(* IEC 61131-3 sources: TrakMap/InstallerSetup/Installer AS Technology Solution/Logical/Source/Diagnostic/TrakDiag, 7 files *)

(* ---- Types.typ ---- *)
TYPE
	VisType : 	STRUCT
		OpenSegDialog : BOOL;
		OpenShuttleDialog : BOOL;
	END_STRUCT;
	CheckStateEnum :
		(
		WAIT_FOR_CHECK,
		READ_DATA,
		READ_DATA_SEG_STATE,
		CHECK_SEG_STATE,
		READ_DATA_SEG_ERROR_STAT,
		CHECK_ERROR_STAT,
		READ_DATA_SEG_ERROR,
		CHECK_ERROR_CODE,
		WRITE_WARNING_CODE,
		READ_DATA_SEG_LAG,
		CHECK_SEG_LAG,
		READ_DATA_SEG_VEL,
		CHECK_SEG_VEL,
		READ_DATA_SEG_TEMP,
		CHECK_DATA_SEG_TEMP,
		WRITE_SPEED_FILTER,
		WRITE_SPEED_FILTER_WAIT,
		WRITE_ZERO_PITCH,
		READ_EXEC_ERROR,
		READ_SEG_STATUS,
		WRITE_SEG_RESET,
		WAIT_FOR_DONE
		);
	SegErrorCheckType : 	STRUCT
		CheckState : CheckStateEnum;
		CmdCheckErrorCode : BOOL;
		DataReadExecutionError : BOOL;
		ErrorNumber : UINT;
		SegStatusBits : UDINT;
		ErrorStatusBit : BOOL;
		ErrorStatus : UDINT;
	END_STRUCT;
	DiagFbsType : 	STRUCT
		Asm : DiagAsmFbsTyp;
		Seg : DiagSegFbsTyp;
	END_STRUCT;
	DiagAsmFbsTyp : 	STRUCT
		ReadInfo : MC_BR_AsmReadInfo_AcpTrak;
		ReadStatus : MC_BR_AsmReadStatus_AcpTrak;
	END_STRUCT;
	DiagSegFbsTyp : 	STRUCT
		ReadInfo : ARRAY[0..NUM_SEG]OF MC_BR_SegReadInfo_AcpTrak;
		ReadStatus : ARRAY[0..NUM_SEG]OF MC_BR_SegReadStatus_AcpTrak;
		ProcessParID : ARRAY[0..NUM_SEG]OF MC_BR_SegProcessParID_AcpTrak;
	END_STRUCT;
END_TYPE

(* ---- CheckErrorCode.st ---- *)
ACTION actCheckErrorCode:

	FOR SegIndex := 0 TO NUM_SEG DO

		CASE SegErrorCheck[SegIndex].CheckState OF

			WAIT_FOR_CHECK:
				//Wait for the command to check the error code ParID on the segment
				DiagFbs.Seg.ProcessParID[SegIndex].Execute := FALSE;

				IF SegErrorCheck[SegIndex].CmdCheckErrorCode THEN
					ErrorCodeIDInfo[SegIndex].DataType := mcACPTRAK_SEG_PARTYPE_UINT;
					ErrorCodeIDInfo[SegIndex].ParID := mcACPPAR_ERROR_NUMBER;
					ErrorCodeIDInfo[SegIndex].VariableAddress := ADR(SegErrorCheck[SegIndex].ErrorNumber);

					DiagFbs.Seg.ProcessParID[SegIndex].Execute := TRUE;
					DiagFbs.Seg.ProcessParID[SegIndex].Segment := ADR(TrakDiag.Seg.SegList[SegIndex].McType);
					DiagFbs.Seg.ProcessParID[SegIndex].ChannelIndex := 0;
					DiagFbs.Seg.ProcessParID[SegIndex].NumberOfParIDs := 1;
					DiagFbs.Seg.ProcessParID[SegIndex].Mode := mcACPTRAK_SEG_PARID_GET_NO_NCT;
					DiagFbs.Seg.ProcessParID[SegIndex].DataAddress := ADR(ErrorCodeIDInfo[SegIndex]);
					SegErrorCheck[SegIndex].CheckState := READ_DATA_SEG_ERROR;
					SegErrorCheck[SegIndex].CmdCheckErrorCode := FALSE; //Reset check command

				END_IF

			READ_DATA_SEG_ERROR:
				//Check for completion of reading the PARID for

				IF DiagFbs.Seg.ProcessParID[SegIndex].Done THEN
					//If the parID was successfully read, go to check error code state
					SegErrorCheck[SegIndex].CheckState := CHECK_ERROR_CODE;
					DiagFbs.Seg.ProcessParID[SegIndex].Execute := FALSE;
					SegErrorCheck[SegIndex].DataReadExecutionError := FALSE;

				ELSIF DiagFbs.Seg.ProcessParID[SegIndex].Error THEN
					//If there was an error in reading, go to error start
					SegErrorCheck[SegIndex].CheckState := READ_EXEC_ERROR;
				END_IF
			CHECK_ERROR_CODE:

				IF (SegErrorCheck[SegIndex].ErrorNumber = 0) OR (SegErrorCheck[SegIndex].ErrorNumber = 36005) THEN
					//Segment has no new error recorded. Shows either 0 or the commanded warning (36005) used to overwrite old errors
					TrakDiag.Seg.SegList[SegIndex].Status.ErrorCode := 0;
					SegErrorCheck[SegIndex].CheckState := WAIT_FOR_CHECK;
					TrakDiag.Seg.SegList[SegIndex].Status.Error := FALSE;

				ELSE
					//Otherwise, there is a new error on this segment
					TrakDiag.Seg.SegList[SegIndex].Status.ErrorCode := SegErrorCheck[SegIndex].ErrorNumber;

					TrakDiag.Seg.SegList[SegIndex].Status.Error := TRUE;
					//Send to overwrite state to store a known error number (36005) in the error code parID
					SegErrorCheck[SegIndex].CheckState := WRITE_WARNING_CODE;

				END_IF
			WRITE_WARNING_CODE:
				//Write commanded warning code (36005) to error parid
				DiagFbs.Seg.ProcessParID[SegIndex].DataAddress := ADR(SegWarningCmdIDInfo);
				DiagFbs.Seg.ProcessParID[SegIndex].ChannelIndex := 0;
				DiagFbs.Seg.ProcessParID[SegIndex].Mode := mcACPTRAK_SEG_PARID_SET;
				DiagFbs.Seg.ProcessParID[SegIndex].NumberOfParIDs := 0;
				DiagFbs.Seg.ProcessParID[SegIndex].Execute := TRUE;

				IF DiagFbs.Seg.ProcessParID[SegIndex].Done THEN
					//return to wait state
					DiagFbs.Seg.ProcessParID[SegIndex].Execute := FALSE;
					SegErrorCheck[SegIndex].CheckState := WAIT_FOR_CHECK;

				ELSIF DiagFbs.Seg.ProcessParID[SegIndex].Error THEN
					SegErrorCheck[SegIndex].CheckState := READ_EXEC_ERROR;
				END_IF
			READ_EXEC_ERROR:
				DiagFbs.Seg.ProcessParID[SegIndex].Execute := FALSE;
				SegErrorCheck[SegIndex].DataReadExecutionError := TRUE;

				IF DiagFbs.Seg.ProcessParID[SegIndex].Error = FALSE THEN
					SegErrorCheck[SegIndex].CheckState := WAIT_FOR_CHECK;
				END_IF
		END_CASE
	DiagFbs.Seg.ProcessParID[SegIndex]();
	END_FOR
END_ACTION

(* ---- Cyclic.st ---- *)
PROGRAM _CYCLIC

	MC_BR_SegCommandError_AcpTrak_0(Segment := ADR(TrakDiag.Seg.SegList[0].McType));

	IF MC_BR_SegCommandError_AcpTrak_0.Done THEN
		MC_BR_SegCommandError_AcpTrak_0.Execute := FALSE;
	END_IF

	(***********************************ASSEMBLY INFORMATION******************************	)
	(*Read Assebly Status*)

	DiagFbs.Asm.ReadStatus.Enable	:= TRUE;
	DiagFbs.Asm.ReadStatus();

	IF DiagFbs.Asm.ReadStatus.Valid THEN
		TrakDiag.Asm.AssemblyDisabled 	:= DiagFbs.Asm.ReadStatus.AssemblyDisabled;
		TrakDiag.Asm.AssemblyErrorStop := DiagFbs.Asm.ReadStatus.AssemblyErrorStop;
		TrakDiag.Asm.AssemblyReady		:= DiagFbs.Asm.ReadStatus.AssemblyReady;
		TrakDiag.Asm.AssemblyHoming	:= DiagFbs.Asm.ReadStatus.AssemblyHoming;
		TrakDiag.Asm.AssemblyStopping	:= DiagFbs.Asm.ReadStatus.AssemblyStopping;
	END_IF

	(*Read Assembly Info *)

	DiagFbs.Asm.ReadInfo.Enable		:= TRUE;
	DiagFbs.Asm.ReadInfo();

	IF DiagFbs.Asm.ReadInfo.Valid THEN
		TrakDiag.Asm.CommunicationReady 	:= DiagFbs.Asm.ReadInfo.AssemblyInfo.CommunicationReady;
		TrakDiag.Asm.PowerOn				:= DiagFbs.Asm.ReadInfo.AssemblyInfo.PowerOn;
		TrakDiag.Asm.ReadyForPowerOn		:= DiagFbs.Asm.ReadInfo.AssemblyInfo.ReadyForPowerOn;
		TrakDiag.Asm.ShuttlesCount 			:= DiagFbs.Asm.ReadInfo.AssemblyInfo.ShuttlesCount;
		TrakDiag.Asm.ShuttleInErrorStopCount := DiagFbs.Asm.ReadInfo.AssemblyInfo.ShuttlesInErrorStopCount;
		TrakDiag.Asm.StartupCount			:= DiagFbs.Asm.ReadInfo.AssemblyInfo.StartupCount;
	END_IF

	(****************************** SEGMENT ERROR INFORMATION *****************************************)

	FOR SegIndex := 0 TO NUM_SEG DO

		IF TrakDiag.Seg.SegList[SegIndex].McType.controlif <> 0 THEN //If the array contains a segment reference

			DiagFbs.Seg.ReadInfo[SegIndex].Segment 	:= ADR(TrakDiag.Seg.SegList[SegIndex].McType);
			DiagFbs.Seg.ReadInfo[SegIndex].Enable	:= TRUE;
			DiagFbs.Seg.ReadInfo[SegIndex]();

			IF DiagFbs.Seg.ReadInfo[SegIndex].Valid THEN
				//Capture Segment Info
				TrakDiag.Seg.SegList[SegIndex].Status.CommunicationReady 	:= DiagFbs.Seg.ReadInfo[SegIndex].SegmentInfo.CommunicationReady;
				TrakDiag.Seg.SegList[SegIndex].Status.ReadyForPowerOn		:= DiagFbs.Seg.ReadInfo[SegIndex].SegmentInfo.ReadyForPowerOn;
				TrakDiag.Seg.SegList[SegIndex].Status.PowerOn				:= DiagFbs.Seg.ReadInfo[SegIndex].SegmentInfo.PowerOn;
				TrakDiag.Seg.SegList[SegIndex].Status.StartupCount			:= DiagFbs.Seg.ReadInfo[SegIndex].SegmentInfo.StartupCount;
				TrakDiag.Seg.SegList[SegIndex].Status.CommunicationState	:= DiagFbs.Seg.ReadInfo[SegIndex].SegmentInfo.CommunicationState;

			END_IF

			DiagFbs.Seg.ReadStatus[SegIndex].Segment := ADR(TrakDiag.Seg.SegList[SegIndex].McType);
			DiagFbs.Seg.ReadStatus[SegIndex].Enable	:= TRUE;
			DiagFbs.Seg.ReadStatus[SegIndex]();

			IF DiagFbs.Seg.ReadStatus[SegIndex].Valid THEN

				//Check for change of state to ErrorStop to command reading error data, IF communication is ready
				IF ((TrakDiag.Seg.SegList[SegIndex].Status.SegmentErrorStop = FALSE AND DiagFbs.Seg.ReadStatus[SegIndex].SegmentErrorStop = TRUE))
					AND (TrakDiag.Seg.SegList[SegIndex].Status.CommunicationReady = TRUE) THEN

					SegErrorCheck[SegIndex].CmdCheckErrorCode := TRUE;

					//Check for change of state from ErrorStop to reset error number in diag structure
				ELSIF ((TrakDiag.Seg.SegList[SegIndex].Status.SegmentErrorStop = TRUE) AND (DiagFbs.Seg.ReadStatus[SegIndex].SegmentErrorStop = FALSE))
					AND (TrakDiag.Seg.SegList[SegIndex].Status.CommunicationReady = TRUE) THEN

					TrakDiag.Seg.SegList[SegIndex].Status.ErrorCode := 0;

				END_IF
				//Capture Segment Status

				TrakDiag.Seg.SegList[SegIndex].Status.SegmentDisabled	:= DiagFbs.Seg.ReadStatus[SegIndex].SegmentDisabled;
				TrakDiag.Seg.SegList[SegIndex].Status.SegmentErrorStop	:= DiagFbs.Seg.ReadStatus[SegIndex].SegmentErrorStop;
				TrakDiag.Seg.SegList[SegIndex].Status.SegmentReady		:= DiagFbs.Seg.ReadStatus[SegIndex].SegmentReady;
				TrakDiag.Seg.SegList[SegIndex].Status.SegmentStopping	:= DiagFbs.Seg.ReadStatus[SegIndex].SegmentStopping;
			END_IF
		END_IF
	END_FOR

	CpuSim := DiagCpuIsSimulated() OR DiagCpuIsARsim();

	IF CpuSim = FALSE THEN
		actCheckErrorCode;
	END_IF

	(***********************************TRAKMAP******************************)

	//Fetch ShuttleUserData Example
	IF EDGEPOS(paperCore.ClickData.Shuttle.Valid) THEN
		MC_BR_ShCopyUserData_AcpTrak_0.Axis         := ADR(paperCore.ClickData.Shuttle.Data.Axis);
		MC_BR_ShCopyUserData_AcpTrak_0.Execute      := TRUE;
		MC_BR_ShCopyUserData_AcpTrak_0.DataAddress  := ADR(ShuttleUserData);
		MC_BR_ShCopyUserData_AcpTrak_0.DataSize     := SIZEOF(ShuttleUserData);
		MC_BR_ShCopyUserData_AcpTrak_0.Mode         := mcACPTRAK_USERDATA_GET;
	END_IF

	paperCore();

	MC_BR_ShCopyUserData_AcpTrak_0();
	MC_BR_ShCopyUserData_AcpTrak_0.Execute := FALSE;

END_PROGRAM

(* ---- Exit.st ---- *)
PROGRAM _EXIT
			(* Insert code here *)

END_PROGRAM

(* ---- Init.st ---- *)
PROGRAM _INIT

	SegDefinition;

	paperCore.SegmentCount := TrakDiag.Seg.SegCount;
	paperCore.Segments := ADR(TrakDiag.Seg.SegList);
	paperCore.Options := ADR(paperOptions);
	paperCore.Enable := TRUE;
	paperCore.Assembly := ADR(DiagInterface.SampleTrak);
	paperCore.ShuttleMon := ADR(DiagInterface.ShuttleMon);
	paperCore.TrakStatus := ADR(TrakDiag);

	paperOptions.Color.Offset := SIZEOF(UDINT);
	paperOptions.Segment.Enabled := TRUE;
	paperOptions.Shuttle.Enabled := TRUE;
	paperOptions.Color.Enabled := TRUE;
END_PROGRAM

(* ---- SegDefinition.st ---- *)
//This file was automatically generated using the TrakMapImporter program. Verify that the segment names and assembly name match your project values correctly
ACTION SegDefinition:
	TrakDiag.Seg.SegList[0].Name  := 'gSeg_A_1';		TrakDiag.Seg.SegList[0].McType := gSeg_A_1;
	TrakDiag.Seg.SegList[1].Name  := 'gSeg_A_2';		TrakDiag.Seg.SegList[1].McType := gSeg_A_2;
	TrakDiag.Seg.SegList[2].Name  := 'gSeg_A_3';		TrakDiag.Seg.SegList[2].McType := gSeg_A_3;
	TrakDiag.Seg.SegList[3].Name  := 'gSeg_A_4';		TrakDiag.Seg.SegList[3].McType := gSeg_A_4;
	TrakDiag.Seg.SegList[4].Name  := 'gSeg_A_5';		TrakDiag.Seg.SegList[4].McType := gSeg_A_5;
	TrakDiag.Seg.SegList[5].Name  := 'gSeg_A_6';		TrakDiag.Seg.SegList[5].McType := gSeg_A_6;
	TrakDiag.Seg.SegList[6].Name  := 'gSeg_A_7';		TrakDiag.Seg.SegList[6].McType := gSeg_A_7;
	TrakDiag.Seg.SegList[7].Name  := 'gSeg_A_8';		TrakDiag.Seg.SegList[7].McType := gSeg_A_8;
	TrakDiag.Seg.SegList[8].Name  := 'gSeg_A_9';		TrakDiag.Seg.SegList[8].McType := gSeg_A_9;
	TrakDiag.Seg.SegList[9].Name  := 'gSeg_A_10';		TrakDiag.Seg.SegList[9].McType := gSeg_A_10;
	TrakDiag.Seg.SegList[10].Name  := 'gSeg_A_11';		TrakDiag.Seg.SegList[10].McType := gSeg_A_11;
	TrakDiag.Seg.SegList[11].Name  := 'gSeg_A_12';		TrakDiag.Seg.SegList[11].McType := gSeg_A_12;

	TrakDiag.Seg.SegList[12].Name  := 'gSeg_B_1';		TrakDiag.Seg.SegList[12].McType := gSeg_B_1;
	TrakDiag.Seg.SegList[13].Name  := 'gSeg_B_2';		TrakDiag.Seg.SegList[13].McType := gSeg_B_2;
	TrakDiag.Seg.SegList[14].Name  := 'gSeg_B_3';		TrakDiag.Seg.SegList[14].McType := gSeg_B_3;
	TrakDiag.Seg.SegList[15].Name  := 'gSeg_B_4';		TrakDiag.Seg.SegList[15].McType := gSeg_B_4;
	TrakDiag.Seg.SegList[16].Name  := 'gSeg_B_5';		TrakDiag.Seg.SegList[16].McType := gSeg_B_5;
	TrakDiag.Seg.SegList[17].Name  := 'gSeg_B_6';		TrakDiag.Seg.SegList[17].McType := gSeg_B_6;
	TrakDiag.Seg.SegList[18].Name  := 'gSeg_B_7';		TrakDiag.Seg.SegList[18].McType := gSeg_B_7;
	TrakDiag.Seg.SegList[19].Name  := 'gSeg_B_8';		TrakDiag.Seg.SegList[19].McType := gSeg_B_8;
	TrakDiag.Seg.SegList[20].Name  := 'gSeg_B_9';		TrakDiag.Seg.SegList[20].McType := gSeg_B_9;
	TrakDiag.Seg.SegList[21].Name  := 'gSeg_B_10';		TrakDiag.Seg.SegList[21].McType := gSeg_B_10;
	TrakDiag.Seg.SegList[22].Name  := 'gSeg_B_11';		TrakDiag.Seg.SegList[22].McType := gSeg_B_11;

	TrakDiag.Seg.SegCount := 23;

	TrakDiag.Seg.SegListAdr := ADR(TrakDiag.Seg.SegList);

	DiagFbs.Asm.ReadInfo.Assembly := ADR(DiagInterface.SampleTrak);
	DiagFbs.Asm.ReadStatus.Assembly := ADR(DiagInterface.SampleTrak);

	paperCore.ViewBoxCfg.MinX := -0.735577;
	paperCore.ViewBoxCfg.MinY := -0.115;
	paperCore.ViewBoxCfg.Width := 2.13115;
	paperCore.ViewBoxCfg.Height := 1.52;

END_ACTION

(* ---- Variables.var ---- *)
VAR
	MC_BR_ShCopyUserData_AcpTrak_0 : MC_BR_ShCopyUserData_AcpTrak;
	ShuttleUserData : ShuttleUserDataType;
	ErrorCodeIDInfo : ARRAY[0..NUM_SEG] OF McAcpTrakSegProcessParIDType;
	SegWarningCmdIDInfo : McAcpTrakSegProcessParIDType;
	SegErrorCheck : ARRAY[0..NUM_SEG] OF SegErrorCheckType;
	CpuSim : BOOL;
END_VAR
(*For testing only*)
VAR
	MC_BR_SegCommandError_AcpTrak_0 : MC_BR_SegCommandError_AcpTrak;
END_VAR
(*Declarations for TrakMap*)
VAR
	paperCore : TrkPaperCore;
	paperOptions : TrkPaperCoreOptionsType;
	TrakDiag : TrkDiagStatusType;
	DiagFbs : DiagFbsType;
	SegIndex : USINT;
END_VAR
